// TwinCAT 3 PLC project Library
// Title: LCLS Sample Delivery
// Company: SLAC - LCLS
// ProjectVersion: 0.0.0
// ProgramVersion: 3.1.4023.0
// libraries:
//   LCLS Vacuum, * (SLAC - LCLS)
//   PMPS, * (SLAC - LCLS)
//   Tc2_EtherCAT, * (Beckhoff Automation GmbH)
//   Tc2_MC2, * (Beckhoff Automation GmbH)
//   Tc2_ModbusSrv, * (Beckhoff Automation GmbH)
//   Tc2_SerialCom, * (Beckhoff Automation GmbH)
//   Tc2_Standard, * (Beckhoff Automation GmbH)
//   Tc2_SUPS, * (Beckhoff Automation GmbH)
//   Tc2_System, * (Beckhoff Automation GmbH)
//   Tc2_Utilities, * (Beckhoff Automation GmbH)
//   Tc3_Module, * (Beckhoff Automation GmbH)
//   TcUnit, * (www.tcunit.org)
//   LCLS General,2.12.0,SLAC
// project tree:
//   DUTs/ALI/ E_AxisMoveMode.TcDUT (not stored), E_CTRL_MODE.TcDUT (not stored), E_PropValveFBState.TcDUT (not stored), HMI_PropValveCtrlState.TcDUT (not stored), ST_ALI.TcDUT (not stored), ST_ManipAxis.TcDUT (not stored), ST_PIDParams.TcDUT (not stored), ST_PressureController.TcDUT (not stored), ST_PropValveMKS253.TcDUT (not stored)
//   DUTs/Bronkhorst/ E_BHElFlowUnit.TcDUT (not stored), ST_BhElFlow.TcDUT (not stored)
//   DUTs/ E_AxisMotionState.TcDUT (not stored), ST_ManifoldValve.TcDUT (not stored), ST_Proportionair.TcDUT (not stored), ST_RegDeadbandControls.TcDUT (not stored), ST_Regulator.TcDUT (not stored), ST_SelectorM3.TcDUT (not stored), ST_Shaker.TcDUT (not stored), ST_ShakerControls.TcDUT (not stored), ST_Strings.TcDUT (not stored)
//   DUTs/General/ E_CTRL_MODE_1.TcDUT (not stored)
//   DUTs/IO_Structs/ ST_ALIIO.TcDUT (not stored), ST_M3DeviceBaseIO.TcDUT (not stored), ST_SerialComm.TcDUT (not stored)
//   DUTs/RCC/ E_RCC_STATES.TcDUT, ST_RCC.TcDUT
//   DUTs/Sensirion/ E_SensirionFMMode.TcTLEO (not stored), ST_SensirionFM.TcDUT (not stored), ST_SensirionFMControl.TcDUT (not stored), ST_SensirionFMStatus.TcDUT (not stored)
//   DUTs/TEC/ ST_TECControl.TcDUT (not stored), ST_TECStatus.TcDUT (not stored)
//   DUTs/Vici/ ST_4PViciValveSampleNames.TcDUT (not stored), ST_ViciControl.TcDUT, ST_ViciStatus.TcDUT (not stored)
//   GVLs/ GVL_SAMPLE.TcGVL (not stored)
//   / PlcTask.TcTTO
//   POUs/ALI/ FB_ALI.TcPOU (not stored), FB_ManipAxis.TcPOU (not stored), FB_PID_EXT.TcPOU (not stored), FB_PropValve.TcPOU (not stored), F_AxisRef_To_MSTA.TcPOU (not stored), MC_SmoothMover.TcPOU (not stored)
//   POUs/Bronkhorst/ FB_BronkhorstMFM.TcPOU (not stored)
//   POUs/DigitalOutput/ FB_SolenoidPair.TcPOU
//   POUs/ EXAMPLE_DEPLOYMENT.TcPOU, PRG_TEST.TcPOU
//   POUs/GasManifold/ FB_GasManifold.TcPOU (not stored), FB_ManiValve.TcPOU (not stored)
//   POUs/Helpers/ FB_EcatDiag.TcPOU (not stored), FB_SelectorSync.TcPOU (not stored), FB_SerialCommWrapper.TcPOU (not stored), FB_ShiftByteArray.TcPOU (not stored)
//   POUs/PCM/ FB_PressureControlModule.TcPOU (not stored)
//   POUs/RCC/ FB_RCC.TcPOU, FB_RCC_SM.TcPOU, FB_VRC_NC_OPNLS.TcPOU
//   POUs/Regulators/ FB_ProportionairRegulator.TcPOU (not stored), FB_Regulator.TcPOU (not stored), F_rPressure.TcPOU (not stored)
//   POUs/Selectors/ FB_SelectorM3.TcPOU (not stored)
//   POUs/Sensirion/ FB_SenserionFlowMeter.TcPOU, FB_SensirionDriver.TcPOU (not stored), FB_SensirionTransaction.TcPOU (not stored), fSHDLCChecksum.TcPOU (not stored)
//   POUs/TEC/ FB_TECDriver.TcPOU (not stored), FB_TECTransaction.TcPOU (not stored)
//   POUs/Tests/ FB_RCC_TEST.TcPOU
//   POUs/VICI/ FB_4PortViciValve.TcPOU (not stored), FB_ViciDriver.TcPOU (not stored), FB_ViciTransaction.TcPOU (not stored), FB_ViciValve.TcPOU
// real-time tasks:
//   TASK PlcTask: cycle T#10ms, priority 20, ADS port 350

CONFIGURATION Library
    RESOURCE PLC ON TwinCAT3
        TASK PlcTask(INTERVAL := T#10ms, PRIORITY := 20);
        PROGRAM PRG_TEST WITH PlcTask : PRG_TEST;
    END_RESOURCE
END_CONFIGURATION

// ---- DUTs/RCC/E_RCC_STATES.TcDUT
{attribute 'qualified_only'}
{attribute 'strict'}
TYPE E_RCC_STATES :
(
    ERROR := -1,
    IDLE := 0,
    INIT := 1,
    OPEN_VRC_02_FOR_T1 := 2,
    DRAIN := 3,
    DRAIN_CHECK := 4,
    OPEN_VRC_01_FOR_T3 := 5,
    OPEN_VRC_04_FOR_T4 := 6
);
END_TYPE

// ---- DUTs/RCC/ST_RCC.TcDUT
TYPE ST_RCC :
STRUCT
    {attribute 'pytmc' :='
        pv: Tinterval
        io: io
    '} // Time before cycle starts
    TInterval : REAL := 10;
    {attribute 'pytmc' :='
        pv: T1
        io: io
    '}
    T1 : REAL := 20;
    {attribute 'pytmc' :='
        pv: T2
        io: io
    '}
    T2 : REAL := 10;
    {attribute 'pytmc' :='
        pv: T3
        io: io
    '}
    T3 : REAL := 5;
    {attribute 'pytmc' :='
        pv: T4
        io: io
    '}
    T4 : REAL := 10;
    {attribute 'pytmc' :=' pv: RUNCLEAN'}
    bRunClean : BOOL := TRUE;

    {attribute 'pytmc' :=' pv: CLEAR_ERROR'}
    bClearError : BOOL := FALSE;
    {attribute 'pytmc' :=' pv: ERROR'}
    bError : BOOL := FALSE;
    {attribute 'pytmc' :=' pv: STOP_CYCLE'}
    bStop : BOOL := FALSE;

    {attribute 'pytmc' :=' pv: START_CYCLE'}
    bStartCycle : BOOL  := FALSE;

    {attribute 'pytmc' :=' pv: ILK_Setpoint '}
    RCC_GCP_01_INTERLOCK_SETPOINT : REAL := 10;
    {attribute 'pytmc' :=' pv: OverrideMode '}
    xSystemOverrideMode_RCC : BOOL := FALSE;

    eCurrentState : INT := E_RCC_STATES.IDLE;

    {attribute 'pytmc' :='
        pv: RCC_RUNNING
        io: o
    '}
    bRunning : BOOL := FALSE;
    {attribute 'pytmc' :='
        pv: RCC_TIMER
        io: o
    '}
    tTimerReadBack : STRING := '';
    {attribute 'pytmc' :=' pv: sLogMessage '}
    sLogMessage : T_MaxString := '';

    RCC_VRC_01_OPEN_OK : BOOL;
    RCC_VRC_02_OPEN_OK : BOOL;
    RCC_VRC_03_OPEN_OK : BOOL;
    RCC_VRC_04_OPEN_OK : BOOL;

END_STRUCT
END_TYPE

// ---- DUTs/Vici/ST_ViciControl.TcDUT
TYPE ST_ViciControl :
STRUCT
    sViciReply			: STRING;
    iReqPos				: INT;
    xDirection			: BOOL;
    iAddress			: INT;
    iPortCount			: INT := 12; // Max Number of Ports Supported by Valve
END_STRUCT
END_TYPE

// ---- POUs/PRG_TEST.TcPOU
PROGRAM PRG_TEST
VAR
    fbRCC_TEST : FB_RCC_TEST;
END_VAR

TcUnit.RUN();

END_PROGRAM

// ---- POUs/Tests/FB_RCC_TEST.TcPOU
FUNCTION_BLOCK FB_RCC_TEST EXTENDS FB_TestSuite
VAR
    fbRCC : FB_RCC;
    stRCC_CTL : ST_RCC;
    stRCC_VRC_01 : ST_VRC;
    stRCC_VRC_02 : ST_VRC;
    stRCC_VRC_03 : ST_VRC;
    stRCC_VRC_04 : ST_VRC;
    stRCC_GCP_01 : ST_VG;
    tTimer1 : TON;
    bInitTest : BOOL := TRUE;
    xSystemOverrideMode_RCC: BOOL := FALSE;

    fbRCC1 : FB_RCC;
    stRCC1_CTL : ST_RCC;
    stRCC_VRC_01_01 : ST_VRC;
    stRCC_VRC_02_01 : ST_VRC;
    stRCC_VRC_03_01 : ST_VRC;
    stRCC_VRC_04_01 : ST_VRC;
    stRCC_GCP_01_01 : ST_VG;
    tTimer1_01 : TON;
    bInitTest_01 : BOOL := TRUE;
    xSystemOverrideMode_RCC_01: BOOL := FALSE;

    fbRCC2 : FB_RCC;
    stRCC2_CTL : ST_RCC;
    stRCC_VRC_01_02 : ST_VRC;
    stRCC_VRC_02_02 : ST_VRC;
    stRCC_VRC_03_02 : ST_VRC;
    stRCC_VRC_04_02 : ST_VRC;
    stRCC_GCP_01_02 : ST_VG;
    tTimer1_02 : TON;
    bInitTest_02 : BOOL := TRUE;
    xSystemOverrideMode_RCC_02: BOOL := FALSE;

    // VARS FOR TestSingleCyleExpectToTransitionThoughOneCycle
    bSeenStateZero : BOOL := FALSE;
    bSeenStateOne : BOOL := FALSE;
    bSeenStateTwo : BOOL := FALSE;
    bSeenStateThree : BOOL := FALSE;
    bSeenStateFour : BOOL := FALSE;
    bSeenStateFive : BOOL := FALSE;

    // VARS FOR TestStopCycleExpectToReturnToIdleState
    iDrainCount : INT := 0;

END_VAR

TestSingleCyleExpectToTransitionThoughOneCycle();
TestErrorExpectToTransitionToErroState();
TestStopCycleExpectToReturnToIdleState();

METHOD TestErrorExpectToTransitionToErroState : REFERENCE TO FB_Test
VAR_INPUT
END_VAR
TEST('TestErrorExpectToTransitionToErroState');

tTimer1_01(IN:=TRUE, PT:=T#46S);

IF bInitTest_01 THEN
    stRCC1_CTL.bStartCycle := TRUE;
    bInitTest_01 := FALSE;
    AssertEquals_INT(Expected:= E_RCC_STATES.IDLE,
        Actual:= stRCC1_CTL.eCurrentState,
        Message:= 'DID NOT START IN IDLE STATE');
END_IF

fbRCC1(stRCC_GCP_01:=stRCC_GCP_01_01,
    stRCC_VRC_01:= stRCC_VRC_01_01,
    stRCC_VRC_02:= stRCC_VRC_02_01,
    stRCC_VRC_03:= stRCC_VRC_03_01,
    stRCC_VRC_04:= stRCC_VRC_04_01,
    stRCC_CTL:= stRCC1_CTL
);


IF stRCC1_CTL.eCurrentState = E_RCC_STATES.DRAIN THEN
    // Enable RCC_VRC_03_OPEN_OK SO WE CAN MOVE ONTO NEXT STATE
    (* Valve can open only when CRIX-RCC-GCP-01 reading < setpoint Torr and CRIX-RCC-VRC-01 and 04 are closed*)
    stRCC_GCP_01_01.rPRESS := 0;
    stRCC_GCP_01_01.xPRESS_OK  := FALSE;
    stRCC_VRC_01_01.i_xClsLS := TRUE;
    stRCC_VRC_01_01.q_xOPN_DO := FALSE;
    stRCC_VRC_04_01.i_xClsLS := TRUE;
    stRCC_VRC_04_01.q_xOPN_DO := FALSE;
 END_IF


IF tTimer1_01.Q OR stRCC1_CTL.bError THEN
    AssertEquals_BOOL(Expected:= stRCC1_CTL.bError ,
        Actual:= TRUE,
        Message:= 'ERROR FLAG NOT SET');

    AssertEquals_INT(Expected:=E_RCC_STATES.ERROR ,
        Actual:= stRCC1_CTL.eCurrentState,
        Message:= 'NOT IN ERROR STATE');

    stRCC1_CTL.bClearError := TRUE; // CLEAR ERRORS

    //CYCLE ONE MORE TIME TO SEE IF ERRORS CLEARD
    fbRCC1(stRCC_GCP_01:=stRCC_GCP_01_01,
        stRCC_VRC_01:= stRCC_VRC_01_01,
        stRCC_VRC_02:= stRCC_VRC_02_01,
        stRCC_VRC_03:= stRCC_VRC_03_01,
        stRCC_VRC_04:= stRCC_VRC_04_01,
        stRCC_CTL := stRCC1_CTL
    );


    AssertEquals_BOOL(Expected:= stRCC1_CTL.bError ,
        Actual:= FALSE,
        Message:= 'ERROR FLAG NOT CLEARD');

    AssertEquals_INT(Expected:=E_RCC_STATES.IDLE ,
        Actual:= stRCC1_CTL.eCurrentState,
        Message:= 'NOT IN IDLE STATE');

    TEST_FINISHED();
    bInitTest_01 := TRUE;
    tTimer1_01(IN:=FALSE, PT:=T#46S);
END_IF
END_METHOD

METHOD TestSingleCyleExpectToTransitionThoughOneCycle : REFERENCE TO FB_Test
VAR_INPUT
END_VAR
VAR
END_VAR
TEST('TestSingleCyleExpectToTransitionThoughOneCycle');

tTimer1(IN:=TRUE, PT:=T#46s);

IF bInitTest THEN
    stRCC_CTL.bStartCycle := TRUE;
    bInitTest := FALSE;
    AssertEquals_INT(Expected:= E_RCC_STATES.IDLE,
        Actual:= stRCC_CTL.eCurrentState,
        Message:= 'DID NOT START AT FIRST STATE');
END_IF

fbRCC(stRCC_GCP_01:=stRCC_GCP_01,
    stRCC_VRC_01:= stRCC_VRC_01,
    stRCC_VRC_02:= stRCC_VRC_02,
    stRCC_VRC_03:= stRCC_VRC_03,
    stRCC_VRC_04:= stRCC_VRC_04,
    stRCC_CTL := stRCC_CTL
);

// CHECK IF WE HAVE SEEN ALL THE STATES
IF stRCC_CTL.eCurrentState = E_RCC_STATES.INIT THEN bSeenStateZero := TRUE; END_IF
IF stRCC_CTL.eCurrentState = E_RCC_STATES.OPEN_VRC_02_FOR_T1 THEN bSeenStateOne := TRUE; END_IF
IF stRCC_CTL.eCurrentState = E_RCC_STATES.DRAIN THEN
    // Enable RCC_VRC_03_OPEN_OK SO WE CAN MOVE ONTO NEXT STATE
    (* Valve can open only when CRIX-RCC-GCP-01 reading < setpoint Torr and CRIX-RCC-VRC-01 and 04 are closed*)
    bSeenStateTwo := TRUE;
    stRCC_GCP_01.rPRESS := 0;
    stRCC_GCP_01.xPRESS_OK  := TRUE;
    stRCC_VRC_01.i_xClsLS := TRUE;
    stRCC_VRC_01.q_xOPN_DO := FALSE;
    stRCC_VRC_04.i_xClsLS := TRUE;
    stRCC_VRC_04.q_xOPN_DO := FALSE;
 END_IF
IF stRCC_CTL.eCurrentState = E_RCC_STATES.DRAIN_CHECK THEN bSeenStateThree := TRUE; END_IF
IF stRCC_CTL.eCurrentState = E_RCC_STATES.OPEN_VRC_01_FOR_T3 THEN bSeenStateFour := TRUE; END_IF
IF stRCC_CTL.eCurrentState = E_RCC_STATES.OPEN_VRC_04_FOR_T4 THEN bSeenStateFive :=TRUE; END_IF

        // THIS IS A TEST


IF tTimer1.Q THEN
    // HAVE SE SEEN ALL STAES?
    AssertEquals_BOOL(Expected:= (bSeenStateZero AND
                                    bSeenStateOne AND
                                    bSeenStateTwo AND
                                    bSeenStateThree AND
                                    bSeenStateFour AND
                                    bSeenStateFive),
        Actual:= TRUE,
        Message:= 'HAVE NOT VISITED ALL STATES');
    TEST_FINISHED();
    bInitTest := TRUE;
    tTimer1(IN:=FALSE, PT:=T#46S);
END_IF
END_METHOD

METHOD TestStopCycleExpectToReturnToIdleState : REFERENCE TO FB_Test
VAR_INPUT
END_VAR
TEST('TestStopCycleExpectToReturnToIdleState');

tTimer1_02(PT:=T#500ms);

IF bInitTest_02 THEN
    stRCC2_CTL.bStartCycle := TRUE;
    bInitTest_02 := FALSE;
    tTimer1_02.IN:=FALSE;
    AssertEquals_INT(Expected:= E_RCC_STATES.IDLE,
        Actual:= stRCC2_CTL.eCurrentState,
        Message:= 'DID NOT START AT FIRST STATE');
END_IF

fbRCC2(	stRCC_GCP_01:= stRCC_GCP_01_02,
        stRCC_VRC_01:= stRCC_VRC_01_02,
        stRCC_VRC_02:= stRCC_VRC_02_02,
        stRCC_VRC_03:= stRCC_VRC_03_02,
        stRCC_VRC_04:= stRCC_VRC_04_02,
        stRCC_CTL := stRCC2_CTL
);

IF stRCC2_CTL.eCurrentState = E_RCC_STATES.DRAIN THEN
    // Enable RCC_VRC_03_OPEN_OK SO WE CAN MOVE ONTO NEXT STATE
    (* Valve can open only when CRIX-RCC-GCP-01 reading < setpoint Torr and CRIX-RCC-VRC-01 and 04 are closed*)
    stRCC_GCP_01_02.rPRESS := 20;
    stRCC_GCP_01_02.xPRESS_OK  := TRUE;
    stRCC_VRC_01_02.i_xClsLS := TRUE;
    stRCC_VRC_01_02.q_xOPN_DO := FALSE;
    stRCC_VRC_04_02.i_xClsLS := TRUE;
    stRCC_VRC_04_02.q_xOPN_DO := FALSE;
    tTimer1_02.IN:=TRUE;
    stRCC2_CTL.bStop := TRUE;
 END_IF


IF tTimer1_02.Q THEN
    AssertEquals_INT(Expected:= E_RCC_STATES.IDLE,
        Actual:= stRCC2_CTL.eCurrentState,
        Message:= 'DID NOT END IN IDLE STATE');
    TEST_FINISHED();
    bInitTest_02 := TRUE;
END_IF
END_METHOD

END_FUNCTION_BLOCK

// ---- POUs/RCC/FB_RCC.TcPOU
FUNCTION_BLOCK FB_RCC
VAR_IN_OUT
    stRCC_VRC_01 : ST_VRC;
    stRCC_VRC_02 : ST_VRC;
    stRCC_VRC_03 : ST_VRC;
    stRCC_VRC_04 : ST_VRC;
    stRCC_GCP_01 : ST_VG;
    stRCC_CTL : ST_RCC;
END_VAR
VAR_OUTPUT
END_VAR
VAR
    fbRCC : FB_RCC_SM; // RCC STATE MATCHINE
    fbFormatString : FB_FormatString;
    TInterval : TIME;
    T1 : TIME;
    T2 : TIME;
    T3 : TIME;
    T4 : TIME;
END_VAR

// convert int to time to seconds
TInterval := REAL_TO_TIME(stRCC_CTL.TInterval * 1E3);
T1 := REAL_TO_TIME(stRCC_CTL.T1 * 1E3);
T2 := REAL_TO_TIME(stRCC_CTL.T2 * 1E3);
T3 := REAL_TO_TIME(stRCC_CTL.T3 * 1E3);
T4 := REAL_TO_TIME(stRCC_CTL.T4 * 1E3);

fbRCC(
    stRCC_VRC_01 := stRCC_VRC_01,
    stRCC_VRC_02 := stRCC_VRC_02,
    stRCC_VRC_03 := stRCC_VRC_03,
    stRCC_VRC_04 := stRCC_VRC_04,
    stRCC_GCP_01 := stRCC_GCP_01,
    TInterval := TInterval,
    T1 := T1,
    T2 := T2,
    T3 := T3,
    T4 := T4,
    bRunClean := stRCC_CTL.bRunClean,
    bClearError := stRCC_CTL.bClearError,
    bError := stRCC_CTL.bError,
    bStop := stRCC_CTL.bStop,
    bStartCycle := stRCC_CTL.bStartCycle,
    tTimerRBV := stRCC_CTL.tTimerReadBack,
    bRunning := stRCC_CTL.bRunning,
    RCC_GCP_01_INTERLOCK_SETPOINT := stRCC_CTL.RCC_GCP_01_INTERLOCK_SETPOINT,
    xSystemOverrideMode_RCC := stRCC_CTL.xSystemOverrideMode_RCC,
    eCurrentState := stRCC_CTL.eCurrentState,
    sLogMessage := stRCC_CTL.sLogMessage,
    RCC_VRC_01_OPEN_OK := stRCC_CTL.RCC_VRC_01_OPEN_OK,
    RCC_VRC_02_OPEN_OK := stRCC_CTL.RCC_VRC_02_OPEN_OK,
    RCC_VRC_03_OPEN_OK := stRCC_CTL.RCC_VRC_03_OPEN_OK,
    RCC_VRC_04_OPEN_OK := stRCC_CTL.RCC_VRC_04_OPEN_OK
    );

END_FUNCTION_BLOCK

// ---- POUs/RCC/FB_RCC_SM.TcPOU
FUNCTION_BLOCK FB_RCC_SM
VAR_IN_OUT
    stRCC_VRC_01 : ST_VRC;
    stRCC_VRC_02 : ST_VRC;
    stRCC_VRC_03 : ST_VRC;
    stRCC_VRC_04 : ST_VRC;
    stRCC_GCP_01 : ST_VG;

    TInterval : TIME; // Time in between cycles
    T1 : TIME;
    T2 : TIME;
    T3 : TIME;
    T4 : TIME;

    bRunClean : BOOL;
    bClearError : BOOL;
    bError : BOOL;
    bStop : BOOL;
    bStartCycle : BOOL;
    bRunning : BOOL;
    tTimerRBV : STRING;

    RCC_GCP_01_INTERLOCK_SETPOINT : REAL;
    xSystemOverrideMode_RCC : BOOL;
    eCurrentState : INT;
    sLogMessage : T_MaxString;

    RCC_VRC_01_OPEN_OK : BOOL;
    RCC_VRC_02_OPEN_OK : BOOL;
    RCC_VRC_03_OPEN_OK : BOOL;
    RCC_VRC_04_OPEN_OK : BOOL;
END_VAR
VAR
    RCC_GCP_ILK_CONV : REAL;
    tTimer1 : TON;
END_VAR

RCC_GCP_ILK_CONV := RCC_GCP_01_INTERLOCK_SETPOINT * 1E2; // Convert to Torr
tTimerRBV := TIME_TO_STRING(tTimer1.ET);

(* Valve can open only when CRIX-RCC-VRC-02 and 03 are closed*)
RCC_VRC_01_OPEN_OK := ( stRCC_VRC_02.i_xClsLS AND NOT stRCC_VRC_02.q_xOPN_DO ) AND
                                    ( stRCC_VRC_03.i_xClsLS AND NOT stRCC_VRC_03.q_xOPN_DO ) ;

(* Valve can open only when CRIX-RCC-VRC-01 and 04 are closed*)
RCC_VRC_02_OPEN_OK := ( stRCC_VRC_01.i_xClsLS AND NOT stRCC_VRC_01.q_xOPN_DO ) AND
                                    ( stRCC_VRC_04.i_xClsLS AND NOT stRCC_VRC_04.q_xOPN_DO );

(* Valve can open only when CRIX-RCC-GCP-01 reading < setpoint Torr and CRIX-RCC-VRC-01 and 04 are closed*)
RCC_VRC_03_OPEN_OK := (stRCC_GCP_01.rPRESS < RCC_GCP_ILK_CONV AND stRCC_GCP_01.xPRESS_OK ) AND
                                 ( stRCC_VRC_01.i_xClsLS AND NOT stRCC_VRC_01.q_xOPN_DO ) AND
                                              ( stRCC_VRC_04.i_xClsLS AND NOT stRCC_VRC_04.q_xOPN_DO );


(* Valve can open only when CRIX-RCC-VRC-02 and 03 are closed*)
RCC_VRC_04_OPEN_OK := ( stRCC_VRC_02.i_xClsLS AND NOT stRCC_VRC_02.q_xOPN_DO ) AND
                                      ( stRCC_VRC_03.i_xClsLS AND NOT stRCC_VRC_03.q_xOPN_DO ) ;


IF bStop THEN
    eCurrentState:= E_RCC_STATES.INIT;
    bStartCycle := FALSE;
END_IF

 CASE eCurrentState OF
    E_RCC_STATES.ERROR: // SOMETHING WENT WRONG
        bRunning := FALSE;
        stRCC_VRC_01.pv_xOPN_SW := FALSE;
        stRCC_VRC_02.pv_xOPN_SW := FALSE;
        stRCC_VRC_03.pv_xOPN_SW := FALSE;
        stRCC_VRC_04.pv_xOPN_SW := FALSE;

        IF bClearError THEN
            eCurrentState := E_RCC_STATES.IDLE;
            bError := FALSE;
            bClearError:= FALSE;
        END_IF

    E_RCC_STATES.IDLE: // -1
        sLogMessage := 'IDLE';
        bRunning := FALSE;
        IF bStartCycle THEN
            tTimer1(IN:=FALSE); // RESTART TIMER
            eCurrentState := E_RCC_STATES.INIT;
            bRunning := TRUE;
        END_IF

    E_RCC_STATES.INIT: // 0
        sLogMessage := 'WAITING FOR CYCLE TO START';
        stRCC_VRC_01.pv_xOPN_SW := FALSE;
        stRCC_VRC_02.pv_xOPN_SW := FALSE;
        stRCC_VRC_03.pv_xOPN_SW := FALSE;
        stRCC_VRC_04.pv_xOPN_SW := FALSE;
        tTimer1(IN:=TRUE, PT:=TInterval);

        IF tTimer1.Q THEN
            eCurrentState:= E_RCC_STATES.OPEN_VRC_02_FOR_T1;
            tTimer1(IN:=FALSE); // RESTART TIMER
        END_IF

        IF bStop THEN
            eCurrentState:= E_RCC_STATES.IDLE;
            bStop := FALSE;
        END_IF

    E_RCC_STATES.OPEN_VRC_02_FOR_T1: // OPEN 1
        sLogMessage := 'OPEN VAVLE 2 FOR T1 SECONDS';
        tTimer1(IN:=TRUE, PT:=T1);
        stRCC_VRC_02.pv_xOPN_SW := TRUE;

        IF tTimer1.Q THEN
            eCurrentState := E_RCC_STATES.DRAIN;
            tTimer1(IN:=FALSE); // RESTART TIMER
        END_IF

     E_RCC_STATES.DRAIN:	// DRAIN_1 2
        // THIS MIGHT CAUSE THE RCC TO STALL IF THIS CONDITION IS NEVER MET
        sLogMessage := 'DRAINING';
        IF (NOT stRCC_GCP_01.xPRESS_OK) THEN
            eCurrentState := E_RCC_STATES.ERROR;
            bError := TRUE;
        END_IF

        IF RCC_VRC_03_OPEN_OK THEN
            IF bRunClean THEN stRCC_VRC_02.pv_xOPN_SW := FALSE; END_IF
            stRCC_VRC_03.pv_xOPN_SW := TRUE;
            eCurrentState := E_RCC_STATES.DRAIN_CHECK;
        END_IF

    E_RCC_STATES.DRAIN_CHECK:	// CHECK IF WE ARE DON DRAINING 3
        tTimer1(IN:=TRUE, PT:=T2);
        sLogMessage := 'OPEN VALVE 3 FOR T2 SECONDS';

        IF tTimer1.Q THEN
            eCurrentState := E_RCC_STATES.OPEN_VRC_01_FOR_T3;
            IF NOT RCC_VRC_03_OPEN_OK THEN eCurrentState := E_RCC_STATES.OPEN_VRC_02_FOR_T1; END_IF
             stRCC_VRC_03.pv_xOPN_SW := FALSE;
            IF NOT bRunClean THEN stRCC_VRC_02.pv_xOPN_SW := FALSE; END_IF
            tTimer1(IN:=FALSE); // RESTART TIMER
        END_IF

     E_RCC_STATES.OPEN_VRC_01_FOR_T3: // OPEN VRC_01 for T3 4
         sLogMessage := 'OPEN VALVE 1 FOR T3 SECONDS';
        tTimer1(IN:=TRUE, PT:=T3);
        stRCC_VRC_01.pv_xOPN_SW := TRUE;
        IF tTimer1.Q THEN
            eCurrentState := E_RCC_STATES.OPEN_VRC_04_FOR_T4;
            tTimer1(IN:=FALSE); // RESTART TIMER
        END_IF

     E_RCC_STATES.OPEN_VRC_04_FOR_T4: // OPEN VRC_04 for T4 5
         sLogMessage := 'OPEN VALVE 4 FOR T4 SECONDS';
        tTimer1(IN:=TRUE, PT:=T4);
        stRCC_VRC_04.pv_xOPN_SW := TRUE;
        IF tTimer1.Q THEN
            sLogMessage := 'CLOSING VALVE 1&4, RESTARTING CYCLE';
            eCurrentState := E_RCC_STATES.IDLE;
            stRCC_VRC_01.pv_xOPN_SW := FALSE;
            stRCC_VRC_04.pv_xOPN_SW := FALSE;
            tTimer1(IN:=FALSE); // RESTART TIMER
        END_IF


END_CASE

END_FUNCTION_BLOCK

// ---- POUs/DigitalOutput/FB_SolenoidPair.TcPOU
FUNCTION_BLOCK FB_SolenoidPair
VAR_INPUT
END_VAR
VAR_OUTPUT
END_VAR
VAR_IN_OUT
END_VAR
VAR
    {attribute 'pytmc' := '
        pv: Valve:01:Open
        io: io
        field: ZNAM "CLOSE"
        field: ONAM "OPEN"
     '}
    q_xDO1 AT %Q*	:	BOOL;
    {attribute 'pytmc' := '
        pv: Valve:02:Open
        io: io
        field: ZNAM "CLOSE"
        field: ONAM "OPEN"
     '}
    q_xDO2 AT %Q*	:	BOOL;

    {attribute 'pytmc' := '
        pv: Switch
        io: o
     '}
    i_xEpics AT %I* : BOOL; // open A when False, open B when True

    {attribute 'pytmc' := '
        pv: Debug
        io: o
     '}
    i_xDebug AT %I* : BOOL; // if True, do not set valves according to i_xEpics
END_VAR

(* If debug, set independently. Else, only open one valve according to i_xEpics *)
IF NOT i_xDebug THEN
    q_xDO1 := NOT i_xEpics;
    q_xDO2 := i_xEpics;
END_IF

END_FUNCTION_BLOCK

// ---- POUs/EXAMPLE_DEPLOYMENT.TcPOU
PROGRAM EXAMPLE_DEPLOYMENT
VAR
{attribute 'pytmc' := 'pv: @(P):SEL:A'}
{attribute 'TcLinkTo' := '.stSensSerial.stComIn.Status := TIIB[M3 Selector A Serial IO (EP6002-0002)]^COM TxPDO-Map Inputs Channel 1^Status;
                          .stViciSerial.stComIn.Status := TIIB[M3 Selector A Serial IO (EP6002-0002)]^COM TxPDO-Map Inputs Channel 2^Status;
                          .stSensSerial.stComOut.Ctrl := TIID^MAIN (EtherCAT)^M3 Selector A Serial IO (EP6002-0002)^COM RxPDO-Map Outputs Channel 1^Ctrl;
                          .stViciSerial.stComOut.Ctrl := TIID^MAIN (EtherCAT)^M3 Selector A Serial IO (EP6002-0002)^COM RxPDO-Map Outputs Channel 2^Ctrl;
                          .stShaker01.q_xPwrDO := TIIB[M3 Selector A Digital IO (EP2338-1001)]^Channel 9^Output;
                          .stShaker02.q_xPwrDO := TIIB[M3 Selector A Digital IO (EP2338-1001)]^Channel 10^Output;
                          .stShaker03.q_xPwrDO := TIIB[M3 Selector A Digital IO (EP2338-1001)]^Channel 11^Output;
                          .stShaker04.q_xPwrDO := TIIB[M3 Selector A Digital IO (EP2338-1001)]^Channel 12^Output;
                          .stBaseIO.i_SyncUnitWC := TIID^MAIN (EtherCAT)^M3 Selector A (EP1111)^WcState^WcState;
'}
fbSelectorA : FB_SelectorM3;

{attribute 'pytmc' := 'pv: @(P):PCM:A'}
{attribute 'TcLinkTo' := '.stPropAir1.i_iPressRB := TIID^MAIN (EtherCAT)^PCM A (EP4374-0002)^AI Inputs Channel 1^Value;
                          .stPropAir2.i_iPressRB := TIID^MAIN (EtherCAT)^PCM A (EP4374-0002)^AI Inputs Channel 2^Value;
                          .stPropAir1.q_iPressCt := TIID^MAIN (EtherCAT)^PCM A (EP4374-0002)^AO Outputs Channel 3^Analog output;
                          .stPropAir2.q_iPressCt := TIID^MAIN (EtherCAT)^PCM A (EP4374-0002)^AO Outputs Channel 4^Analog output;
                          .stSerial1.stComIn.Status := TIID^MAIN (EtherCAT)^PCM A (EP6002-0002)^COM TxPDO-Map Inputs Channel 1^Status;
                          .stSerial2.stComIn.Status := TIID^MAIN (EtherCAT)^PCM A (EP6002-0002)^COM TxPDO-Map Inputs Channel 2^Status;
                          .stSerial1.stComOut.Ctrl := TIID^MAIN (EtherCAT)^PCM A (EP6002-0002)^COM RxPDO-Map Outputs Channel 1^Ctrl;
                          .stSerial2.stComOut.Ctrl := TIID^MAIN (EtherCAT)^PCM A (EP6002-0002)^COM RxPDO-Map Outputs Channel 2^Ctrl;
                          .stBaseIO.i_SyncUnitWC := TIID^MAIN (EtherCAT)^PCM A (EP1111)^WcState^WcState;
'}
fbPCMA		: FB_PressureControlModule;

{attribute 'pytmc' := 'pv: @(P):MAN'}
{attribute 'TcLinkTo' := '.stValve[1].qxDO := TIIB[Gas_Mani_ValveCtrl (EP2338-0001)]^Channel 9^Output;
                          .stValve[1].ixOPN := TIIB[Gas_Mani_ValveRbk (EP2338-0001)]^Channel 1^Input;
                          .stValve[2].qxDO := TIIB[Gas_Mani_ValveCtrl (EP2338-0001)]^Channel 10^Output;
                          .stValve[2].ixOPN := TIIB[Gas_Mani_ValveRbk (EP2338-0001)]^Channel 2^Input;
                          .stValve[3].qxDO := TIIB[Gas_Mani_ValveCtrl (EP2338-0001)]^Channel 11^Output;
                          .stValve[3].ixOPN := TIIB[Gas_Mani_ValveRbk (EP2338-0001)]^Channel 3^Input;
                          .stValve[4].qxDO := TIIB[Gas_Mani_ValveCtrl (EP2338-0001)]^Channel 12^Output;
                          .stValve[4].ixOPN := TIIB[Gas_Mani_ValveRbk (EP2338-0001)]^Channel 4^Input;
                          .stValve[5].qxDO := TIIB[Gas_Mani_ValveCtrl (EP2338-0001)]^Channel 13^Output;
                          .stValve[5].ixOPN := TIIB[Gas_Mani_ValveRbk (EP2338-0001)]^Channel 5^Input;
                          .stValve[6].qxDO := TIIB[Gas_Mani_ValveCtrl (EP2338-0001)]^Channel 14^Output;
                          .stValve[6].ixOPN := TIIB[Gas_Mani_ValveRbk (EP2338-0001)]^Channel 6^Input;
                          .stValve[7].qxDO := TIIB[Gas_Mani_ValveCtrl (EP2338-0001)]^Channel 15^Output;
                          .stValve[7].ixOPN := TIIB[Gas_Mani_ValveRbk (EP2338-0001)]^Channel 7^Input;
                          .stBaseIO.i_SyncUnitWC :=	TIID^MAIN (EtherCAT)^Gas_Mani (EP1111)^WcState^WcState;
'}
fbGasMan : FB_GasManifold;

{attribute 'pytmc' := 'pv: @(P):MFM:A'}
{attribute 'TcLinkTo' := '.stMFM.i_rFlow := TIID^MAIN (EtherCAT)^Bronkhorst MFM A^TxPDO Map^fMeasure;
                          .stMFM.q_rSetpoint := TIID^MAIN (EtherCAT)^Bronkhorst MFM A^RxPDO Map^fSetpoint;
'}
fbBronkhorstA : FB_BronkhorstMFM;

{attribute 'pytmc' := 'pv: @(P):SPR:A'}
{attribute 'TcLinkTo' := '.q_xDO1 := TIIB[Solenoid Pair A Digital IO (EP2338-0001)]^Channel 9^Output;
                          .q_xDO2 := TIIB[Solenoid Pair A Digital IO (EP2338-0001)]^Channel 10^Output;
'}
fbSolenoidPairA : FB_SolenoidPair;

END_VAR

fbSelectorA();
fbPCMA();
fbGasMan();
fbBronkhorstA();
fbSolenoidPairA();

(* Following execution of all the programs, set the first pass false *)
g_xFirstPass := FALSE;

END_PROGRAM

// ---- POUs/RCC/FB_VRC_NC_OPNLS.TcPOU
(* This Function Block Implements Basic Functionality for ChemRIX NC valve, which has one NC LS mounting at Open position.
This function block is interloked by an input (i_xExtILK_OK). This is so developers can interface with custom
interlocking logic outside this function block.*)
(* Note Interlock Logic is External *)
{attribute 'no_check'}
FUNCTION_BLOCK FB_VRC_NC_OPNLS EXTENDS FB_Valve
VAR_IN_OUT

END_VAR
VAR_INPUT
    i_xExtILK_OK : BOOL; //Connect to Interlock logic condition(e.g F_TURBO_VRC_ILK Function), otherwise, Set to True if the valve is not interlocked
    i_xOverrideMode : BOOL; (*To be linked to global override bit. This Overrides Vacuum logic only, EPS, MPS and PMPS are still enforces*)
END_VAR
VAR_OUTPUT
    {attribute 'pytmc' := '
    pv:
    '}
    iq_stValve : ST_VRC;
END_VAR
VAR
    {attribute 'instance-path'}
    {attribute 'noinit'}
    sPath: STRING;
    xFirstPass	:	BOOL;
    fbFSInit		:	R_TRIG;
    tonOvrd	:	TON;
    tonDelOK : TON;
    rtOK	:	R_TRIG;
    tOvrd	:	TIME := T#10s;
    (* Timeouts*)
    tTimeOutDuration: TIME:= T#30S;
    tOPNtimeout: TON;
    tCLStimeout:TON;
    i_xClsLS : BOOL;


    (*IO*)
    i_xOpnLS	AT%I*: BOOL;
    q_xOPN_DO	AT%Q*: BOOL;

END_VAR


ACT_IO();

(* On first PLC pass, put valve into vented state, which implies a closed valve *)
fbFSInit( CLK := TRUE, Q => xFirstPass);
IF xFirstPass THEN
    iq_stValve.eVGC_State := Vented;
    iq_stValve.pv_xOPN_SW := FALSE;
    ePrevState := INVALID;
END_IF


IF iq_stValve.i_xOpnLS AND iq_stValve.q_xOPN_DO THEN
    iq_stValve.eState:=OPEN;
ELSIF NOT iq_stValve.i_xOpnLS AND NOT iq_stValve.q_xOPN_DO THEN
    iq_stValve.eState:=CLOSED;
END_IF

(*evaluate Valve open external interlock*)
iq_stValve.xOPN_OK := i_xExtILK_OK;
iq_stValve.xEXT_OK := i_xExtILK_OK;
IF NOT iq_stValve.xOPN_OK and NOT tonOvrd.Q THEN
    iq_stValve.pv_xOPN_SW := FALSE;
    iq_stValve.eVGC_State := ERR_ExtFault;
END_IF

IF (iq_stValve.q_xOPN_DO) AND (iq_stValve.xOPN_OK) THEN
    iq_stValve.eVGC_State := AtVacuum;
END_IF


(* Override logic *)
(* Goal: give ability to override, but do so in a way that people won't forget it.
Solution: Override only after ten seconds of override, protect against blips,
when the valve permission goes true for more than ten seconds consistently, remove override
*)

tonDelOK(IN:=iq_stValve.xOPN_OK, PT:=T#10S);
rtOK(CLK:=tonDelOK.Q);
IF rtOK.Q AND iq_stValve.pv_xOvrdOpn THEN
    iq_stValve.pv_xOvrdOpn :=FALSE;
    if (iq_stValve.eState=OPEN) AND (i_xOverrideMode) THEN iq_stValve.pv_xOPN_SW := TRUE; END_IF
    //Log
    fbLogger(sMsg:='Override expired', eSevr:=TcEventSeverity.Warning);
END_IF
// Release the Force Open bit when the system override is false
IF NOT(i_xOverrideMode) THEN  iq_stValve.pv_xOvrdOpn :=FALSE; END_IF
//Override timer
tonOvrd(IN:=iq_stValve.pv_xOvrdOpn, PT:=tOvrd);

(* Here's where the valve opens *)
iq_stValve.q_xOPN_DO := (iq_stValve.pv_xOPN_SW AND iq_stValve.xOPN_OK) OR (tonOvrd.Q AND i_xOverrideMode);


///Check valve moving position timout
IF NOT iq_stValve.i_xClsLS AND tCLStimeout.Q THEN
    iq_stValve.bErrorPresent := TRUE;
    iq_stValve.sErrorMessage := ' Close Timeout';
ELSIF iq_stValve.i_xClsLS AND tOPNtimeout.Q THEN
    iq_stValve.bErrorPresent := TRUE;
    iq_stValve.sErrorMessage := ' Open Timeout';
END_IF

IF (iq_stValve.eState=INVALID) THEN
    iq_stValve.bErrorPresent := TRUE;
    iq_stValve.sErrorMessage := CONCAT(sPath,' Invalid Valve Position');
END_IF

(*Timers*)
tOPNtimeout(IN:= iq_stValve.q_xOPN_DO, PT := tTimeOutDuration );
tCLStimeout(IN:= NOT iq_stValve.q_xOPN_DO, PT := tTimeOutDuration);




// Log States and triggers
ACT_Logger();

ACTION ACT_IO:
(*inputs*)
iq_stValve.i_xOpnLS := 	i_xOpnLS;
iq_stValve.i_xClsLS := i_xClsLS := NOT i_xOpnLS;
iq_stValve.xOverrideMode := i_xOverrideMode;
(*outputs*)
q_xOPN_DO:= iq_stValve.q_xOPN_DO;
END_ACTION

ACTION ACT_Logger:
// ILK logger

IF NOT i_xExtILK_OK AND ePrevState = OPEN THEN
         fbLogger(sMsg:='Lost external interlock while valve was open.', eSevr:=TcEventSeverity.Critical);
END_IF


//STATE Logger

IF ePrevState <> iq_stValve.eState THEN
      CASE iq_stValve.eState OF
        INVALID:
            fbLogger(sMsg:='Valve invalid position.', eSevr:=TcEventSeverity.Critical);
          MOVING:
            fbLogger(sMsg:='Valve moving', eSevr:=TcEventSeverity.Warning);
        OPEN:
            fbLogger(sMsg:='Valve Open.', eSevr:=TcEventSeverity.Info);
        CLOSED:
            fbLogger(sMsg:='Valve closed.', eSevr:=TcEventSeverity.Info);
      END_CASE
      ePrevState := iq_stValve.eState;
  END_IF



// Log valve timeouts
tErrorPresent(CLK:=iq_stValve.bErrorPresent);
IF tErrorPresent.Q THEN fbLogger(sMsg:=iq_stValve.sErrorMessage, eSevr:=TcEventSeverity.Warning); END_IF

// Log valve open
tAction(CLK:= iq_stValve.q_xOPN_DO);
IF tAction.Q THEN fbLogger(sMsg:='Valve commanded open', eSevr:=TcEventSeverity.Info); END_IF

// Log override mode enabled
tOverrideActivated(CLK:= (tonOvrd.Q AND i_xOverrideMode));
IF tOverrideActivated.Q THEN fbLogger(sMsg:='Valve override mode activated', eSevr:=TcEventSeverity.Warning); END_IF
END_ACTION

END_FUNCTION_BLOCK

// ---- POUs/Sensirion/FB_SenserionFlowMeter.TcPOU
FUNCTION_BLOCK FB_SenserionFlowMeter
VAR_INPUT
END_VAR
VAR_OUTPUT
END_VAR
VAR

    {attribute 'pytmc' := 'pv:'}
    astSelFM	: ST_SensirionFM;

    {attribute 'pytmc' := 'pv: Label'}
    sLabel : STRING;

    afbSensirionDriver	: FB_SensirionDriver;

    fbSensSerial : FB_SerialCommWrapper;
    stSensSerial : ST_SerialComm; // Holds Data


END_VAR


astSelFM.stCtrl.xReset := astSelFM.xFMReset;
astSelFM.stCtrl.xCalMode := astSelFM.xFMModeReq;
astSelFM.stCtrl.bAdr := 0;

afbSensirionDriver(
    i_xExecute:= TRUE,
    i_tTimeOut:= t#1s,
    iq_stSerialRXBuffer:= stSensSerial.RxBuffer,
    iq_stSerialTXBuffer:= stSensSerial.TxBuffer,
    q_stStatus=>astSelFM.stStat,
    i_stControl:=astSelFM.stCtrl);

IF afbSensirionDriver.q_xDone OR
    afbSensirionDriver.q_xError OR
    afbSensirionDriver.q_xTimeout THEN

    astSelFM.rFlow := astSelFM.stStat.rFlow;
    astSelFM.xFMOoR := astSelFM.stStat.xOoR;
    astSelFM.xFlowValid := astSelFM.stStat.xFlowValid;
    astSelFM.eFMState := astSelFM.stStat.iState;
    astSelFM.xFMModeRb := astSelFM.stStat.xFMMode;

    (* reset function for next time *)
    afbSensirionDriver.Reset();

END_IF

fbSensSerial(stSerialComm := stSensSerial);

END_FUNCTION_BLOCK

// ---- POUs/VICI/FB_ViciValve.TcPOU
FUNCTION_BLOCK FB_ViciValve
(* FB for VICI RS-232 Valave*)

VAR_INPUT
    iAddress : INT;
    iNumOfPorts : INT;
    iReqPos : INT;
END_VAR
VAR_OUTPUT
END_VAR
VAR
    fbViciDriver  : FB_ViciDriver;
    fbViciSerial  : FB_SerialCommWrapper;
    stViciSerial  : ST_SerialComm;
    stViciVlvCtrl : ST_ViciControl;
    stViciVlvStatus : ST_ViciStatus;

END_VAR

stViciVlvCtrl.iReqPos := iReqPos;
stViciVlvCtrl.iAddress := iAddress;
stViciVlvCtrl.iPortCount := iNumOfPorts;

fbViciDriver(
    i_xExecute:= TRUE,
    i_tTimeOut:= t#10s,
    i_stControl:= stViciVlvCtrl,
    iq_stSerialRXBuffer:= stViciSerial.RxBuffer,
    iq_stSerialTXBuffer:= stViciSerial.TxBuffer,
    q_stStatus=> stViciVlvStatus);

IF 	fbViciDriver.q_xDone OR
    fbViciDriver.q_xError OR
    fbViciDriver.q_xTimeout THEN
    (* reset function for next time *)
    fbViciDriver(i_xExecute:=FALSE,
        iq_stSerialRXBuffer:= stViciSerial.RxBuffer,
        iq_stSerialTXBuffer:= stViciSerial.TxBuffer);

END_IF

fbViciSerial(stSerialComm := stViciSerial);

END_FUNCTION_BLOCK
